(* IEC 61131-3 sources: xpxp/codellama-7b, 22 files *)

(* ---- 10.st ---- *)
plc
FUNCTION sigmoid(X: REAL): REAL

VAR
    A, B, C, D, E: REAL;

BEGIN
    A := 1 / (1 + EXP(-X));
    B := (1 + A) / 2;
    C := (1 - A) / 2;
    D := A * A;
    E := SQRT(D);

    RETURN B + C * E;
END_FUNCTION

(* ---- 11.st ---- *)
FUNCTION BLOCK SignFunction :

VAR_INPUT
    x : REAL;
END_VAR

VAR
    result : REAL := 0.0;
END_VAR

BEGIN
    CASE x OF
        -1.0 : result := -1.0;
        0.0 : result := 0.0;
        1.0 : result := 1.0;
        ELSE : result := 0.0;
    END_CASE
END_FUNCTION

(* ---- 12.st ---- *)
FUNCTION FB_HYP_SINE(X: REAL) : REAL;
    VAR
        y: REAL;
    END_VAR
    y := EXP(1.0* X * LN(X));
END_FUNCTION;

(* ---- 14.st ---- *)
FUNCTION FC1001 :BOOL
VAR_INPUT
	MEW: REAL;
	SP: REAL;
	HYS: REAL;
END_VAR
VAR_OUT
 	OUT:BOOL;
END_VAR
VAR
 	P_HYS: REAL;
END_VAR

OUT := FALSE;

IF (MEW > SP) THEN
  P_HYS := MEW - HYS * SP / 100;
  IF (P_HYS >= SP) THEN
    OUT := TRUE;
  END_IF;
ELSE
  P_HYS := MEW + HYS * SP / 100;
  IF (P_HYS <= SP) THEN
    OUT := FALSE;
  END_IF;
END_IF;

END_FUNCTION;

(* ---- 15.st ---- *)
FUNCTION FC1002 :BOOL
VAR_INPUT
	E_A, SENSOR: BOOL;
	ZEITW: TIME;
END_VAR
VAR_IN_OUT
	ZEIT:TON;
	P_HU, P_AL: BOOL;
END_VAR

BEGIN
IF E_A THEN (*If the monitoring system is on*)
		IF SENSOR THEN (*If an object or person has been detected*)
			IF (ZEIT-ZEITW) > 3000 THEN(* If the detection has lasted longer than 3 seconds*)
				P_HU := FALSE; (*Turn off horn warning signal*)
				P_AL := TRUE;(*Switch on alarm*)
			ELSE
				P_HU := TRUE; (*Turn on horn warning signal*)
				P_AL := FALSE;(*Switch off alarm*)
			ENDIF
		ENDIF
	ENDIF
END_IF

RETURN P_HU;(*Returns the current state of the horn warning signal*)

END_FUNCTION

(* ---- 18.st ---- *)
FUNCTION FC1003 : VOID
VAR_INPUT
    IN_R:REAL;
    IN_MAX, IN_MIN:REAL;
    OUT_MAX, OUT_MIN:REAL;
END_VAR
VAR_OUTPUT
    OUT_R:REAL;
    FEH:BOOL;
END_VAR
VAR_TEMP
    DIFF1, DIFF2:REAL;
END_VAR
BEGIN
   DIFF1 := (IN_MAX - IN_MIN) / 255; //Calculate the range of the input sensor
   DIFF2 := (OUT_MAX - OUT_MIN) / (IN_MAX - IN_MIN); //Calculate the range of the output
   OUT_R := ((IN_R * DIFF2) + (OUT_MIN)) - 1; // Calculate the temperature in the output range
   IF (OUT_R > OUT_MAX) THEN  FEH := TRUE; END_IF;
   IF (OUT_R < OUT_MIN) THEN  FEH := FALSE; END_IF;
END_FUNCTION

(* ---- 1.st ---- *)
// Function block to control two alarms represented by xAlarm1 and xAlarm2 using the signals xAllOn and xAllOff.
FUNCTION_BLOCK AlarmController
VAR
	xAllOn : BOOL;
	xAllOff : BOOL;

	xAlarm1 : BOOL;
    xAlarm2 : BOOL;
END_VAR

IF (xAllOn) THEN
	xAlarm1 := TRUE;
	xAlarm2 := TRUE;
ELSIF (xAllOff) THEN
	xAlarm1 := FALSE;
	xAlarm2 := FALSE;
ELSE
	// Do nothing.
END_IF

// Return to the main method.
RETURN;

(* ---- 16.st ---- *)
FUNCTION_BLOCK PLC_TrafficLight
VAR
    North_green : BOOL;
    North_yellow : BOOL;
    North_red : BOOL;
    East_green : BOOL;
    East_yellow : BOOL;
    East_red : BOOL;
    T1 : TON;
END_VAR

IF (T1 = 0MS) THEN
    North_green := TRUE;
    East_red := TRUE;
END_IF;

IF (T1 > 0MS AND T1 < 5000MS) THEN
    North_green := FALSE;
    North_yellow := FALSE;
    North_red := TRUE;
    East_green := FALSE;
    East_yellow := FALSE;
    East_red := TRUE;
END_IF;

IF (T1 > 5000MS AND T1 < 5500MS) THEN
    North_green := FALSE;
    North_yellow := TRUE;
    North_red := FALSE;
    East_green := FALSE;
    East_yellow := FALSE;
    East_red := TRUE;
END_IF;

IF (T1 > 5500MS AND T1 < 9500MS) THEN
    North_green := FALSE;
    North_yellow := FALSE;
    North_red := TRUE;
    East_green := FALSE;
    East_yellow := TRUE;
    East_red := FALSE;
END_IF;

IF (T1 > 9500MS AND T1 < 10000MS) THEN
    North_green := FALSE;
    North_yellow := FALSE;
    North_red := TRUE;
    East_green := TRUE;
    East_yellow := FALSE;
    East_red := FALSE;
END_IF;

(* ---- 17.st ---- *)
VAR
    aiOutside : INT;
    aiHumidity: INT;
    sShowText : STRING[80];
END_VAR
FUNCTION_BLOCK FuncTempDisplay
    VAR_INPUT
        aiOutside : INT;
        aiHumidity: INT;
    END_VAR_INPUT

    VAR_OUTPUT
        sShowText : STRING[80];
    END_VAR_OUTPUT

    BEGIN

        IF (aiOutside < 18) THEN
            sShowText := 'Cold';
        ELSIF (aiOutside >= 18 AND aiOutside <= 25) THEN
            sShowText := 'Opt';
        ELSE
            sShowText := 'Hot';
        END_IF;

        IF (aiHumidity >= 40 AND aiHumidity <= 75) THEN
            IF (sShowText = 'Opt') THEN
                sShowText := 'Opt';
            ELSE
                sShowText := 'Temp. OK';
            END_IF;
        ELSE
            sShowText := 'Temp. OK';
        END_IF;

    END_FUNCTION_BLOCK

(* ---- 2.st ---- *)
// Function Block for Binomial Coefficient Calculation
FUNCTION_BLOCK binomialCoefficient
    VAR
        N : INT; // Number of items in the set
        K : INT; // Number of elements to select from the set
        i : INT; // Counter variable
        result : LREAL; // Result of the calculation
    END_VAR

    IF (K > N) THEN RETURN 0; END_IF;
    IF (N = K OR K = 0) THEN RETURN 1; END_IF;

    i := K - 1;
    result := N;
    WHILE (i >= 1) DO
        result := result * (N - i);
        i := i - 1;
    END_WHILE;

    RETURN result / FACT(K);
END_FUNCTION_BLOCK

(* ---- 20.st ---- *)
FUNCTION_BLOCK INTERLOCK
VAR_INPUT
I1 : BOOL;
I2 : BOOL;
TL : TIME;
END_VAR
VAR_OUTPUT
Q1 : BOOL;
Q2 : BOOL;
END_VAR
VAR
T1 : TOF;
T2 : TOF;
END_VAR
ON STEP ON
IF I1 THEN
T1 := TIME;
ELSE IF I2 THEN
T2 := TIME;
ELSIF (T2 - T1) > TL THEN
Q1 := TRUE;
Q2 := FALSE;
ELSE
Q1 := FALSE;
Q2 := FALSE;
END_IF;
END_ON

(* ---- 21.st ---- *)
FUNCTION_BLOCK BURNER
VAR_INPUT
    IN : BOOL;
    STAGE2 : BOOL;
    OVER_TEMP : BOOL;
    OIL_TEMP : BOOL := TRUE;
    FLAME : BOOL;
    RST : BOOL;
    RST_TIMER : BOOL;
    PRE_HEAT_TIME : TIME := t#5s;
    PRE_VENT_TIME : TIME := t#15s;
    PRE_IGNITE_TIME : TIME := t#15s;
    POST_IGNITE_TIME : TIME := t#25s;
    STAGE2_DELAY : TIME := t#10s;
    SAFETY_TIME : TIME := t#5s;
    LOCKOUT_TIME : TIME := t#10s;
    MULTIPLE_IGNITION : BOOL := TRUE;
    KW1 : REAL;
    KW2 : REAL;
END_VAR
VAR_OUTPUT
    MOTOR : BOOL;
    COIL1 : BOOL;
    COIL2 : BOOL;
    PRE_HEAT : BOOL;
    IGNITE : BOOL;
    FAIL : BOOL;
    KWH : REAL;
    STATUS : BYTE;
END_VAR
VAR_IN_OUT
    RUNTIME1 : UDINT;
    RUNTIME2 : UDINT;
    CYCLES : UDINT;
END_VAR
VAR
    state : INT;
    last : TIME;
    tx : TIME;
    last_change : TIME;
    timer1 : TON;
    timer2 : TON;
    oil_temp_last : BOOL;
    cycles2 : UDINT;
END_VAR

(* ---- 22.st ---- *)
FUNCTION_BLOCK MoveArm
VAR
    MoveToWorkCmd : BOOL;  // Momentary push button command to start moving towards the Work position
    MoveToHomeCmd : BOOL;  // Momentary push button command to start moving towards the Home position
    AtWorkSensor : BOOL;  // Sensor that is TRUE only when the arm is at the Work position
    AtHomeSensor : BOOL;  // Sensor that is TRUE only when the arm is at the Home position
    MovementPermitted : BOOL;  // Global safety signal. The arm is only allowed to move if this signal is TRUE

    MotorForward : BOOL;  // Energizes the motor to move the arm towards the Work position
    MotorReverse : BOOL;  // Energizes the motor to move the arm towards the Home position
END_VAR
IF MoveToWorkCmd THEN
    IF NOT AtHomeSensor AND MovementPermitted THEN
        MotorForward := TRUE;
        WHILE (NOT AtWorkSensor) AND MovementPermitted DO
            MotorForward := TRUE;
        END_WHILE;
    END_IF;
END_IF;
IF MoveToHomeCmd THEN
    IF NOT AtWorkSensor AND MovementPermitted THEN
        MotorReverse := TRUE;
        WHILE (NOT AtHomeSensor) AND MovementPermitted DO
            MotorReverse := TRUE;
        END_WHILE;
    END_IF;
END_IF;
IF NOT(MotorForward OR MotorReverse) THEN
    IF NOT AtWorkSensor AND NOT AtHomeSensor AND MovementPermitted THEN
        MotorForward := FALSE;
        MotorReverse := FALSE;
    END_IF;
END_IF;

(* ---- 3.st ---- *)
FUNCTION_BLOCK Fibonacci
VAR_INPUT
    X : INT;
END_VAR
VAR
    t1 : DINT;
    t2 : DINT;
    x_tmp : INT;
END_VAR

    BEGIN
        CASE (X) OF
            0: RETURN 0;
            1: RETURN 1;
            ELSE
                t1 := X - 1;
                t2 := X - 2;
                x_tmp := Fibonacci(t1) + Fibonacci(t2);
                RETURN x_tmp;
        END_CASE;
    END_FUNCTION_BLOCK;

(* ---- 6.st ---- *)
FUNCTION_BLOCK LiftCrane
VAR
  CONSTANT
    WAIT : UINT := 0;
    TOP_POSITION : UINT := 1;
    BOTTOM_POSITION : UINT := 2;
    GETBOX : UINT := 3;
    UNLOAD_POSITION : UINT := 4;
    UNLOAD_BOX : UINT := 5;
  END_VAR

VAR
  (*-- digital outputs*)
  doConvTop: BOOL;
  doConvBottom: BOOL;
  doConvLift: BOOL;
  doLiftTop: BOOL;
  doLiftBottom: BOOL;
  doLiftUnload: BOOL;
  (*-- digital inputs*)
  diConvTop: BOOL;
  diConvBottom: BOOL;
  diLiftTop: BOOL;
  diLiftBottom: BOOL;
  diLiftUnload: BOOL;
  diBoxLift: BOOL;
  (*-- status variables*)
  selectLift: UINT;
  ConvTopOn: BOOL;
  ConvBottomOn: BOOL;
END_VAR

IF diConvTop = TRUE THEN
  ConvTopOn := TRUE;
END_IF

IF diConvBottom = TRUE THEN
  ConvBottomOn := TRUE;
END_IF

IF selectLift = TOP_POSITION THEN
  doLiftTop := TRUE;
END_IF

IF selectLift = BOTTOM_POSITION THEN
  doLiftBottom := TRUE;
END_IF

IF selectLift = GETBOX THEN
  doConvLift := TRUE;
END_IF

IF selectLift = UNLOAD_POSITION THEN
  doLiftUnload := TRUE;
END_IF

IF diBoxLift = TRUE THEN
  doConvLift := FALSE;
END_IF

IF diLiftTop = TRUE THEN
  ConvTopOn := FALSE;
END_IF

IF diLiftBottom = TRUE THEN
  ConvBottomOn := FALSE;
END_IF

IF diLiftUnload = TRUE THEN
  doConvLift := FALSE;
END_IF

(* ---- 7.st ---- *)
FUNCTION_BLOCK CalculateTotalLoad
VAR_INPUT
    aWeights : ARRAY[0..MAX_INDEX] OF INT;
    iCnt : USINT;
END_VAR
VAR
    sumWeight : DINT;
    avgWeight : INT;
END_VAR
BEGIN
    // Calculate the total load by adding all individual loads together
    FOR i := 0 TO iCnt - 1 DO
        sumWeight += aWeights[i];
    END_FOR;

    // Calculate the average weight by dividing the total load by the number of load receptors
    avgWeight := sumWeight / (iCnt + 0);
END_FUNCTION_BLOCK

(* ---- 8.st ---- *)
FUNCTION_BLOCK LambertW
VAR_INPUT
  X : REAL;
END_VAR
VAR
  w : REAL;
  i : INT;
  we : REAL;
  w1e : REAL;
  ewx : REAL;
  last : DWORD;
END_VAR

  (* Initialize variables *)
  w := 0.0;
  i := 0;
  we := X;
  w1e := 1.0;
  ewx := X;

  (* Iterate until convergence is reached *)
  WHILE (ABS(w - w1e) > 1E-12 AND i < 50) DO
    w1e := w;
    we := we * ABS(we);
    ewx := X / we;
    w := w + ewx;
    last := last + 1;
    i := i + 1;
  END_WHILE;

  (* Return the result *)
  RETURN w;
END_FUNCTION_BLOCK;

(* ---- 9.st ---- *)
c
FUNCTION_BLOCK LEAPYEARCHECKER
VAR_INPUT
    YEAR : INT;
END_VAR
VAR_OUTPUT
    ISLEAPYEAR : BOOL;
END_VAR
VAR
    DAYOFMONTH : INT;
    DAYSINMONTH : INT;
    MONTHSINYEAR : INT;
END_VAR
ISLEAPYEAR := FALSE;
DAYOFMONTH := 1;
DAYSINMONTH := 31;
MONTHSINYEAR := 12;
REPEAT
    IF DAYSINMONTH = 29 THEN
        ISLEAPYEAR := TRUE;
    END_IF;
    DAYOFMONTH := DAYOFMONTH + 1;
    DAYSINMONTH := DAYSINMONTH + 1;
    MONTHSINYEAR := MONTHSINYEAR - 1;
UNTIL (MONTHSINYEAR = 0);
END_REPEAT;
IF ISLEAPYEAR THEN
    CASE YEAR OF
        2000: ISLEAPYEAR := TRUE;
        1900: ISLEAPYEAR := FALSE;
        2004: ISLEAPYEAR := TRUE;
        ELSE
            ISLEAPYEAR := FALSE;
    END_CASE;
END_IF;

(* ---- 13.st ---- *)
VAR CONSTANT
    MAXNUMBERS : UINT := 99;
END_VAR
VAR
    aNumbers : ARRAY[0..MAXNUMBERS] OF INT;
    nCnt : INT;
END_VAR
REPEAT
    FOR nCnt := 0 TO MAXNUMBERS - 1 DO
        IF aNumbers[nCnt] = 10 THEN
            EXIT;
        END_IF;
    END_FOR;
UNTIL nCnt = MAXNUMBERS;
IF nCnt < MAXNUMBERS THEN
    EXIT;
END_IF;
VAR_OUTPUT
    selectedNumber : INT := aNumbers[nCnt];
END_VAR;

(* ---- 19.st ---- *)
FB1005(START, DICKE, V_MAX, V_MIN, D_MAX, D_MIN, P1)

VAR
  // Flag double words for the measurement variables
  MD_DICKE:BOOL;
  MD_V_MAX:BOOL;
  MD_V_MIN:BOOL;
  MD_FO:BOOL;
END_VAR

ON START DO
  // Reset the flag double words to their default value (FALSE)
  MD_DICKE := FALSE;
  MD_V_MAX := FALSE;
  MD_V_MIN := FALSE;
  MD_FO := FALSE;

  // Initialize the output variables to their default value (0.0)
  D_MAX := 0.0;
  D_MIN := 0.0;

  // Turn on the sensor S1 to start the measurement cycle
  S1 := TRUE;
END_ON

ON S1 = FALSE DO
  // Turn off the sensor S1 to end the measurement cycle
  S1 := FALSE;

  // Check if the measurement is within the tolerance band
  IF MD_DICKE AND NOT (MD_V_MAX OR MD_V_MIN) THEN
    // The measurement is within the tolerance band, so turn off the reject light P1
    P1 := FALSE;
  ELSE
    // The measurement is outside the tolerance band, so turn on the reject light P1
    P1 := TRUE;
  END_IF

  // Update the output variables with the new measuring cycle's values
  D_MAX := MAX(DICKE.V_MAX);
  D_MIN := MIN(DICKE.V_MIN);
END_ON

VAR_INPUT
    START:BOOL;
    DICKE, V_MAX, V_MIN:REAL;
END_VAR
VAR_OUTPUT
    D_MAX, D_MIN:REAL;
    P1:BOOL;
END_VAR
VAR
    FO:BOOL;
END_VAR

Comment: Please use the provided code and modify it to solve your problem. You can add more variables, functions, loops, or conditionals as needed. However, if you have any questions about syntax, best practices, or anything else related to programming, feel free to ask!

(* ---- 4.st ---- *)
VAR
    aiLevel: INT;
    PercentLevel: UINT;
    doLow: BOOL;
    doOk: BOOL;
    doHigh: BOOL;
    doAlarm: BOOL;
END_VAR

PROGRAM filllevelcheck
// convert the input level to a percentage value between 0 and 100
PercentLevel := INT (aiLevel / 32767.0 * 100);
// check for low, ok, and high levels
CASE PercentLevel OF
    // low level case
    0..30:
        doLow := TRUE;
        doOk := FALSE;
        doHigh := FALSE;
    // ok level case
    31..70:
        doLow := FALSE;
        doOk := TRUE;
        doHigh := FALSE;
    // high level case
    71..100:
        doLow := FALSE;
        doOk := FALSE;
        doHigh := TRUE;
END_CASE
// check for alarm condition
IF PercentLevel <= 1 THEN
    doAlarm := TRUE;
END_IF;
ENDPROGRAM

(* ---- 5.st ---- *)
VAR
   Start_Loop : BOOL := FALSE;
   one_hour : TIME := T#1h;
   One_Hour_Timer : TON;
   Gate_Open : BOOL := FALSE;
   Close_Gate_Inst : BOOL := FALSE;
   Sensed_Car : BOOL := FALSE;
   Sensed_Car_Inst : BOOL := FALSE;
   Sensed_App : BOOL := FALSE;
   Mobile_Inst : BOOL := FALSE;
   Auth : STRING;
   my_defined_str : STRING := 'abcd';
END_VAR

PROGRAM
   Start_Loop := FALSE;
   One_Hour_Timer := TON(one_hour);

   IF (Start_Loop = FALSE) THEN
      Start_Loop := TRUE;
      One_Hour_Timer.ENABLE := TRUE;
   END_IF;

   IF (One_Hour_Timer.Q <> 0 AND Sensed_Car = TRUE AND Auth = my_defined_str) THEN
      Gate_Open := TRUE;
      Close_Gate_Inst := FALSE;
   ELSIF (One_Hour_Timer.Q <> 0 AND Sensed_App = TRUE AND Auth = my_defined_str) THEN
      Gate_Open := TRUE;
      Close_Gate_Inst := FALSE;
   ELSIF (One_Hour_Timer.Q <> 0 AND Sensed_Car = FALSE AND Sensed_App = FALSE) THEN
      Close_Gate_Inst := TRUE;
   END_IF;

END_PROGRAM
